// TIA Portal V19 export
DATA_BLOCK "AO SCALING DB"   // DB6
{ S7_Optimized_Access := 'TRUE' }
// stored: MemoryReserve 100
   VAR
      SET : Struct
         "MFG VESSEL MOTOR SPEED" : Real;
         "PREMIXING VESSEL MOTOR SPEED" : Real;
         "STORAGE VESSEL-1 MOTOR SPEED" : Real;
         "STORAGE VESSEL-2 MOTOR SPEED" : Real;
         "SUGAR VESSEL MOTOR SPEED" : Real;
         "AO SPARE_1" : Real;
         "AO SPARE_2" : Real;
         "AO SPARE_3" : Real;
      END_STRUCT;
   END_VAR
   VAR RETAIN
      MIN : Struct
         "MFG VESSEL MOTOR SPEED" : Real;
         "PREMIXING VESSEL MOTOR SPEED" : Real;
         "STORAGE VESSEL-1 MOTOR SPEED" : Real;
         "STORAGE VESSEL-2 MOTOR SPEED" : Real;
         "SUGAR VESSEL MOTOR SPEED" : Real;
         "AO SPARE_1" : Real;
         "AO SPARE_2" : Real;
         "AO SPARE_3" : Real;
      END_STRUCT;
      MAX : Struct
         "MFG VESSEL MOTOR SPEED" : Real;
         "PREMIXING VESSEL MOTOR SPEED" : Real;
         "STORAGE VESSEL-1 MOTOR SPEED" : Real;
         "STORAGE VESSEL-2 MOTOR SPEED" : Real;
         "SUGAR VESSEL MOTOR SPEED" : Real;
         "AO SPARE_1" : Real;
         "AO SPARE_2" : Real;
         "AO SPARE_3" : Real;
      END_STRUCT;
   END_VAR
   VAR
      PV : Struct
         "MFG VESSEL MOTOR SPEED" : Real;
         "PREMIXING VESSEL MOTOR SPEED" : Real;
         "STORAGE VESSEL-1 MOTOR SPEED" : Real;
         "STORAGE VESSEL-2 MOTOR SPEED" : Real;
         "SUGAR VESSEL MOTOR SPEED" : Real;
         "AO SPARE_1" : Real;
         "AO SPARE_2" : Real;
         "AO SPARE_3" : Real;
      END_STRUCT;
   END_VAR
BEGIN
END_DATA_BLOCK
